SUBAPPLICATION Uebung_039_sub_Outputs (* Spiegelabfolge V2 mit Schrittkette SUB Out *)
  (* Standard: 61499-2; Description: Copyright (c) 2024 Meisterschulen am Ostbahnhof This program and the accompanying materials are made available under the terms of the Eclipse Public License 2.0 which is available at https://www.eclipse.org/legal/epl-2.0/ SPDX-License-Identifier: EPL-2.0 *)
  (* Version 1.0, 2024-03-03, Franz Höpfinger, Meisterschulen am Ostbahnhof *)
  PACKAGE Uebungen;
  IMPORT isobus::UT::Q::const::IDs::ID_NULL;
  IMPORT logiBUS::io::DQ::logiBUS_DO;
  IMPORT logiBUS::io::DQ::logiBUS_DO_S;
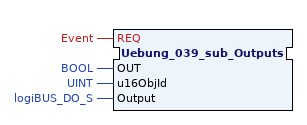
  EVENT_INPUT
    REQ; (* Service Request *)
  END_EVENT
  VAR_INPUT
    OUT : BOOL; (* Output data to resource *)
    u16ObjId : UINT := ID_NULL; (* Object ID Softkey/Button *)
    Output : logiBUS::io::DQ::logiBUS_DO_S := logiBUS_DO::Invalid;
  END_VAR
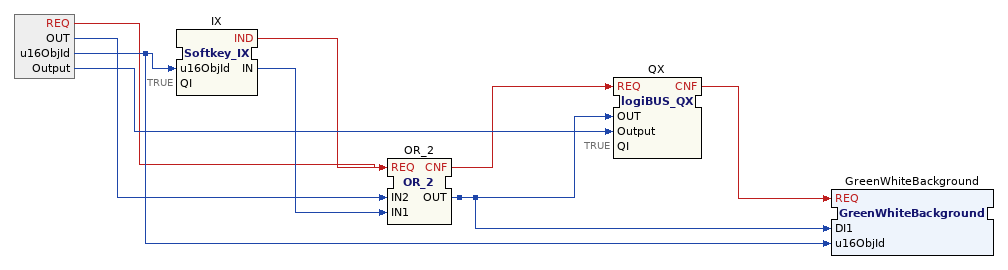
  FBS
    QX : logiBUS::io::DQ::logiBUS_QX(QI := TRUE);
    IX : isobus::UT::io::Softkey::Softkey_IX(QI := TRUE);
    OR_2 : iec61131::bitwiseOperators::OR_2;
  END_FBS
  SUBAPPS
    GreenWhiteBackground : MyLib::sys::GreenWhiteBackground;
  END_SUBAPPS
  EVENT_CONNECTIONS
    OR_2.CNF TO QX.REQ;
    IX.IND TO OR_2.REQ;
    REQ TO OR_2.REQ;
    QX.CNF TO GreenWhiteBackground.REQ;
  END_CONNECTIONS
  DATA_CONNECTIONS
    OUT TO OR_2.IN2;
    IX.IN TO OR_2.IN1;
    OR_2.OUT TO QX.OUT;
    OR_2.OUT TO GreenWhiteBackground.DI1;
    u16ObjId TO GreenWhiteBackground.u16ObjId;
    u16ObjId TO IX.u16ObjId;
    Output TO QX.Output;
  END_CONNECTIONS
END_SUBAPPLICATION
